% RSLogix 500 project Limoneira_2_Line_BiCarb_Original_Backup_Aug_16_2021.RSS, saved by version 11.00.00.00 %
PROJECT "UNTITLED"    % processor: MicroLogix 1200 %

PROGRAM FILES
  LAD 2   19 rungs

DATA FILES
  O0 OUTPUT  4 elements
  I1 INPUT  4 elements
  S2 STATUS  66 elements
  B3 BINARY  1 elements
  T4 TIMER  18 elements
  C5 COUNTER  1 elements
  R6 CONTROL  1 elements
  N7 INTEGER  1 elements
  F8 FLOAT  1 elements

LADDER 2
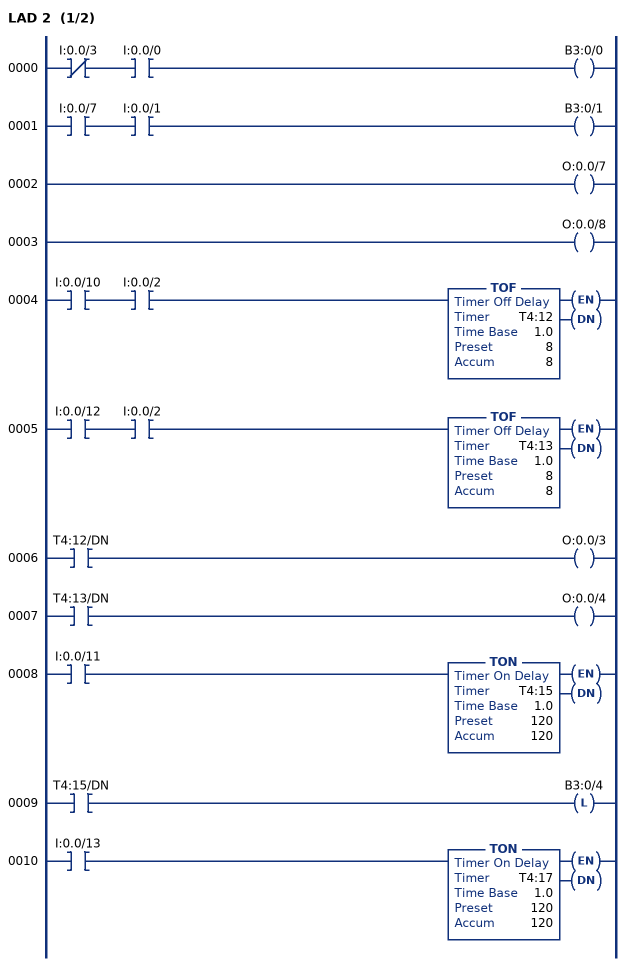
% Rung: 0 %
SOR XIO I:0.0/3 XIC I:0.0/0 OTE B3:0/0 EOR
% Rung: 1 %
SOR XIC I:0.0/7 XIC I:0.0/1 OTE B3:0/1 EOR
% Rung: 2 %
SOR OTE O:0.0/7 EOR
% Rung: 3 %
SOR OTE O:0.0/8 EOR
% Rung: 4 %
SOR XIC I:0.0/10 XIC I:0.0/2 TOF T4:12 1.0 8 8 EOR
% Rung: 5 %
SOR XIC I:0.0/12 XIC I:0.0/2 TOF T4:13 1.0 8 8 EOR
% Rung: 6 %
SOR XIC T4:12/DN OTE O:0.0/3 EOR
% Rung: 7 %
SOR XIC T4:13/DN OTE O:0.0/4 EOR
% Rung: 8 %
SOR XIC I:0.0/11 TON T4:15 1.0 120 120 EOR
% Rung: 9 %
SOR XIC T4:15/DN OTL B3:0/4 EOR
% Rung: 10 %
SOR XIC I:0.0/13 TON T4:17 1.0 120 120 EOR

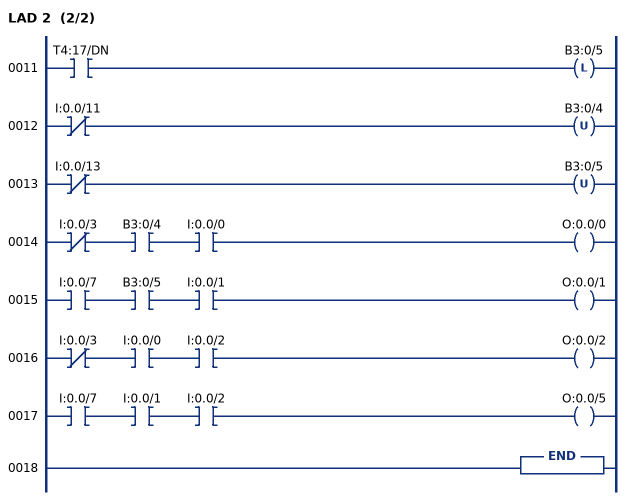
% Rung: 11 %
SOR XIC T4:17/DN OTL B3:0/5 EOR
% Rung: 12 %
SOR XIO I:0.0/11 OTU B3:0/4 EOR
% Rung: 13 %
SOR XIO I:0.0/13 OTU B3:0/5 EOR
% Rung: 14 %
SOR XIO I:0.0/3 XIC B3:0/4 XIC I:0.0/0 OTE O:0.0/0 EOR
% Rung: 15 %
SOR XIC I:0.0/7 XIC B3:0/5 XIC I:0.0/1 OTE O:0.0/1 EOR
% Rung: 16 %
SOR XIO I:0.0/3 XIC I:0.0/0 XIC I:0.0/2 OTE O:0.0/2 EOR
% Rung: 17 %
SOR XIC I:0.0/7 XIC I:0.0/1 XIC I:0.0/2 OTE O:0.0/5 EOR
% Rung: 18 %
SOR END EOR

DATA TABLE (non-zero values as saved)
DATA B3
% B3:0 % 0X0033
DATA T4
% .PRE .ACC %
% T4:0 % 4 0
% T4:1 % 150 150
% T4:2 % 5 0
% T4:3 % 10 0
% T4:10 % 60 0
% T4:11 % 60 0
% T4:12 % 8 8
% T4:13 % 8 8
% T4:15 % 120 120
% T4:16 % 120 0
% T4:17 % 120 120
